Fanuc KAREL source: AVL_POS_NUM.kl

PROGRAM T
%NOLOCKGROUP
VAR
 v0 : INTEGER
 v1 : INTEGER
 v2 : INTEGER
BEGIN
 AVL_POS_NUM(v0, v1, v2)
END T
